// TIA Portal V20 export
DATA_BLOCK "CentralShifter_DB"   // DB31
// stored: InstanceOfName CentralShifter, InstanceOfType FB
"CentralShifter"
   // VAR_INPUT
   //    QR_Reader : DInt;
   // END_VAR
   // VAR
   //    MC_POWER_CS_PP { S7_SetPoint := 'True'} : MC_POWER;
   //    MC_POWER_CS_PL { S7_SetPoint := 'True'} : MC_POWER;
   //    MC_POWER_CS_TP { S7_SetPoint := 'True'} : MC_POWER;
   //    MC_POWER_CS_TL { S7_SetPoint := 'True'} : MC_POWER;
   //    MC_POWER_CS_Virtual { S7_SetPoint := 'True'} : MC_POWER;
   //    MC_RESET_CS_PP { S7_SetPoint := 'True'} : MC_RESET;
   //    MC_RESET_CS_PL { S7_SetPoint := 'True'} : MC_RESET;
   //    MC_RESET_CS_TP { S7_SetPoint := 'True'} : MC_RESET;
   //    MC_RESET_CS_TL { S7_SetPoint := 'True'} : MC_RESET;
   //    MC_GEARIN_CS_PP { S7_SetPoint := 'True'} : MC_GEARIN;
   //    MC_GEARIN_CS_PL { S7_SetPoint := 'True'} : MC_GEARIN;
   //    MC_GEARIN_CS_TP { S7_SetPoint := 'True'} : MC_GEARIN;
   //    MC_GEARIN_CS_TL { S7_SetPoint := 'True'} : MC_GEARIN;
   //    MC_HOME_CS_PP { S7_SetPoint := 'True'} : MC_HOME;
   //    MC_HOME_CS_PL { S7_SetPoint := 'True'} : MC_HOME;
   //    MC_HOME_CS_TP { S7_SetPoint := 'True'} : MC_HOME;
   //    MC_HOME_CS_TL { S7_SetPoint := 'True'} : MC_HOME;
   //    MC_RESET_CS_Virtual { S7_SetPoint := 'True'} : MC_RESET;
   //    MC_MOVEJOG_CS_PL { S7_SetPoint := 'True'} : MC_MOVEJOG;
   //    MC_HOME_CS_Virtual { S7_SetPoint := 'True'} : MC_HOME;
   //    MC_MOVEJOG_CS_PP { S7_SetPoint := 'True'} : MC_MOVEJOG;
   //    MC_MOVEJOG_CS_TL { S7_SetPoint := 'True'} : MC_MOVEJOG;
   //    MC_MOVEJOG_CS_TP { S7_SetPoint := 'True'} : MC_MOVEJOG;
   //    MC_MOVEJOG_CS_Virtual { S7_SetPoint := 'True'} : MC_MOVEJOG;
   //    MC_MOVERELATIVE_CS_Virtual { S7_SetPoint := 'True'} : MC_MOVERELATIVE;
   //    MC_MOVEABSOLUTE_CS_Virtual { S7_SetPoint := 'True'} : MC_MOVEABSOLUTE;
   //    Homeing_Status { S7_SetPoint := 'True'} : Int;
   //    Jog_Backward_Home : Bool;
   //    Jog_Forward_Home : Bool;
   //    Jog_Velocity : Int;
   //    CentralShifter_Auto_Instance { S7_SetPoint := 'True'} : "CentralShifter_AutoDrive";
   //    Jog_Speed { S7_SetPoint := 'True'} : Real;
   //    Auto_Forward : Bool;
   //    Auto_Backward : Bool;
   //    Auto_Turn_OFF { S7_SetPoint := 'True'} : TON_TIME;
   //    CentralShifter_SideShifters_Instance { S7_SetPoint := 'True'} : "CentralShifter_SideShifters";
   //    Position_To_Side_Drive { S7_SetPoint := 'True'} : Bool;
   //    Deceleration : Real;
   //    Arrived_Pos : Int;
   //    CS_Velocity { S7_SetPoint := 'True'} : MC_MOVEVELOCITY;
   //    CentralShifter_Move_Pallets_Instance { S7_SetPoint := 'True'} : "CentralShifter_Move_Pallets";
   //    prevBusy_Jog { S7_SetPoint := 'True'} : Bool;
   //    MC_SETSENSOR_Instance { S7_SetPoint := 'True'} : MC_SETSENSOR;
   //    prevPower { S7_SetPoint := 'True'} : Bool;
   //    Status_Power_Synch : Bool;
   //    Positions_Central : Array[7..13] of DInt;
   //    Central_Auto_Control_Instance { S7_SetPoint := 'True'} : "Central_Auto_Control";
   //    tPowerCheck { S7_SetPoint := 'True'} : TON_TIME;
   //    SinaParaS_CS_M_PL { S7_SetPoint := 'True'} : SinaParaS;
   //    SinaParaS_CS_M_PP { S7_SetPoint := 'True'} : SinaParaS;
   //    SinaParaS_CS_M_TL { S7_SetPoint := 'True'} : SinaParaS;
   //    SinaParaS_CS_M_TP { S7_SetPoint := 'True'} : SinaParaS;
   //    Active_Alarm { S7_SetPoint := 'True'} : Byte;
   //    MC_GEARINVELOCITY_pp { S7_SetPoint := 'True'} : MC_GEARINVELOCITY;
   //    MC_GEARINVELOCITY_tl { S7_SetPoint := 'True'} : MC_GEARINVELOCITY;
   //    MC_GEARINVELOCITY_tp { S7_SetPoint := 'True'} : MC_GEARINVELOCITY;
   //    MC_GEARINVELOCITY_pl { S7_SetPoint := 'True'} : MC_GEARINVELOCITY;
   //    TorqueFB_TEL750_PP { S7_SetPoint := 'True'} : "TorqueFB_TEL750";
   // END_VAR
BEGIN
   CentralShifter_SideShifters_Instance.Stations[12].RL_H3_Pos := 13515;
   CentralShifter_SideShifters_Instance.Stations[13].RL_H3_Pos := 13500;
   CentralShifter_SideShifters_Instance.Stations[12..13].RR_H3_Pos := 13525;
   CentralShifter_SideShifters_Instance.Stations[12].RL_Mid_Pos := 7932;
   CentralShifter_SideShifters_Instance.Stations[13].RL_Mid_Pos := 7916;
   CentralShifter_SideShifters_Instance.Stations[12].RR_Mid_Pos := 7932;
   CentralShifter_SideShifters_Instance.Stations[13].RR_Mid_Pos := 7939;
   CentralShifter_SideShifters_Instance.Stations[12].RL_H5_Pos := 1924;
   CentralShifter_SideShifters_Instance.Stations[13].RL_H5_Pos := 1918;
   CentralShifter_SideShifters_Instance.Stations[12].RR_H5_Pos := 1934;
   CentralShifter_SideShifters_Instance.Stations[13].RR_H5_Pos := 1915;
   CentralShifter_SideShifters_Instance.Stations[12].Correction := 10;
   CentralShifter_SideShifters_Instance.Stations[13].Correction := 15;
END_DATA_BLOCK
